Yaskawa INFORM job: s2D_Face_diagonal.JBI

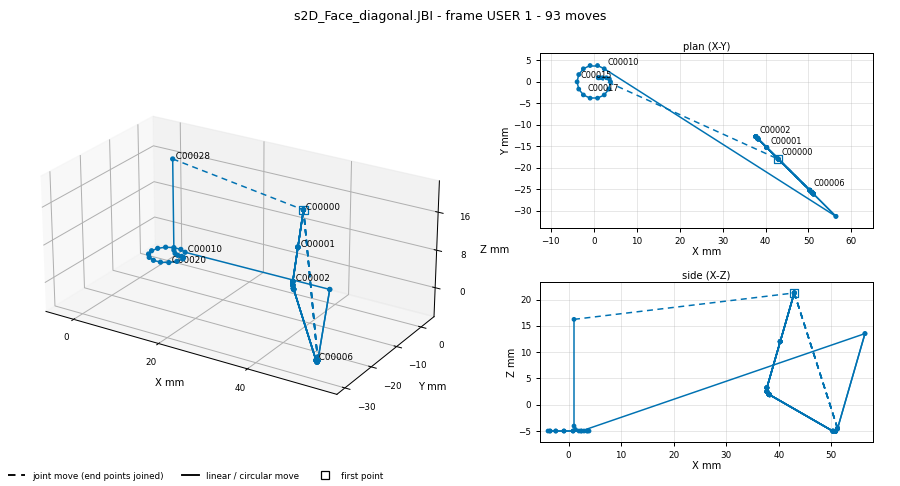
[picture p0: tool path of s2D_Face_diagonal.JBI in frame USER 1, 93 of 93 moves have a stored position in this frame; points joined in program order, loops and branches not executed]
/JOB
//NAME s2D_Face_diagonal
//POS
///NPOS 10,0,0,0,0,0
///USER 1
///TOOL 2
///POSTYPE USER
///RECTAN
///RCONF 1,0,0,0,0,0
C00000=53.984,-29.817,15.539,-90.000,-150.794,-116.565
C00001=53.984,-24.817,6.879,-90.000,-150.794,-116.565
C00002=53.984,-20.744,-0.175,-90.000,-150.794,-116.565
C00003=53.705,-20.407,-0.758,-90.000,-150.794,-116.565
C00004=53.031,-20.268,-1.000,-90.000,-150.794,-116.565
C00005=-55.536,-20.268,-1.000,-90.000,-150.794,-116.565
C00006=-56.209,-20.407,-0.758,-90.000,-150.794,-116.565
C00007=-56.488,-20.744,-0.175,-90.000,-150.794,-116.565
C00008=-56.488,-29.817,15.539,-90.000,-150.794,-116.565
C00000=-54.817,-31.806,15.539,180.000,-152.507,146.310
C00001=-49.817,-31.806,6.879,180.000,-152.507,146.310
C00002=-45.903,-31.806,0.100,180.000,-152.507,146.310
C00003=-45.454,-31.434,-0.678,180.000,-152.507,146.310
C00004=-45.268,-30.536,-1.000,180.000,-152.507,146.310
C00005=-45.268,32.000,-1.000,180.000,-152.507,146.310
C00006=-45.454,32.898,-0.678,180.000,-152.507,146.310
C00007=-45.903,33.270,0.100,180.000,-152.507,146.310
C00008=-54.817,33.270,15.539,180.000,-152.507,146.310
C00000=-54.817,-31.488,15.539,180.000,-152.507,146.310
C00001=-49.817,-31.488,6.879,180.000,-152.507,146.310
C00002=-45.744,-31.488,-0.175,180.000,-152.507,146.310
C00003=-45.407,-31.209,-0.758,180.000,-152.507,146.310
C00004=-45.268,-30.536,-1.000,180.000,-152.507,146.310
C00005=-45.268,32.000,-1.000,180.000,-152.507,146.310
C00006=-45.407,32.674,-0.758,180.000,-152.507,146.310
C00007=-45.744,32.952,-0.175,180.000,-152.507,146.310
C00008=-54.817,32.952,15.539,180.000,-152.507,146.310
C00000=-57.952,29.817,15.539,90.000,-150.794,63.435
C00001=-57.952,24.817,6.879,90.000,-150.794,63.435
C00002=-57.952,20.744,-0.175,90.000,-150.794,63.435
C00003=-57.674,20.407,-0.758,90.000,-150.794,63.435
C00004=-57.000,20.268,-1.000,90.000,-150.794,63.435
C00005=54.657,20.268,-1.000,90.000,-150.794,63.435
C00006=55.330,20.407,-0.758,90.000,-150.794,63.435
C00007=55.609,20.744,-0.175,90.000,-150.794,63.435
C00008=55.609,29.817,15.539,90.000,-150.794,63.435
C00000=-57.952,29.817,15.539,90.000,-150.794,63.435
C00001=-57.952,24.817,6.879,90.000,-150.794,63.435
C00002=-57.952,20.744,-0.175,90.000,-150.794,63.435
C00003=-57.674,20.407,-0.758,90.000,-150.794,63.435
C00004=-57.000,20.268,-1.000,90.000,-150.794,63.435
C00005=54.657,20.268,-1.000,90.000,-150.794,63.435
C00006=55.330,20.407,-0.758,90.000,-150.794,63.435
C00007=55.609,20.744,-0.175,90.000,-150.794,63.435
C00008=55.609,29.817,15.539,90.000,-150.794,63.435
C00000=1.040,-0.952,16.240,0.000,-180.000,-30.000
C00001=1.040,-0.952,6.080,0.000,-180.000,-30.000
C00002=1.040,-0.952,2.000,0.000,-180.000,-30.000
C00003=1.040,-0.952,-4.048,0.000,-180.000,-30.000
C00004=1.319,-0.952,-4.721,0.000,-180.000,-30.000
C00005=1.993,-0.952,-5.000,0.000,-180.000,-30.000
C00006=2.945,-0.952,-5.000,0.000,-180.000,-30.000
C00007=3.619,-0.674,-5.000,0.000,-180.000,-30.000
C00008=3.898,0.000,-5.000,0.000,-180.000,-30.000
C00009=3.512,1.691,-5.000,0.000,-180.000,-30.000
C00010=2.430,3.047,-5.000,0.000,-180.000,-30.000
C00011=0.867,3.800,-5.000,0.000,-180.000,-30.000
C00012=-0.867,3.800,-5.000,0.000,-180.000,-30.000
C00013=-2.430,3.047,-5.000,0.000,-180.000,-30.000
C00014=-3.512,1.691,-5.000,0.000,-180.000,-30.000
C00015=-3.898,0.000,-5.000,0.000,-180.000,-30.000
C00016=-3.512,-1.691,-5.000,0.000,-180.000,-30.000
C00017=-2.430,-3.047,-5.000,0.000,-180.000,-30.000
C00018=-0.867,-3.800,-5.000,0.000,-180.000,-30.000
C00019=0.867,-3.800,-5.000,0.000,-180.000,-30.000
C00020=2.430,-3.047,-5.000,0.000,-180.000,-30.000
C00021=3.512,-1.691,-5.000,0.000,-180.000,-30.000
C00022=3.898,0.000,-5.000,0.000,-180.000,-30.000
C00023=3.619,0.674,-5.000,0.000,-180.000,-30.000
C00024=2.945,0.952,-5.000,0.000,-180.000,-30.000
C00025=1.993,0.952,-5.000,0.000,-180.000,-30.000
C00026=1.319,0.952,-4.721,0.000,-180.000,-30.000
C00027=1.040,0.952,-4.048,0.000,-180.000,-30.000
C00028=1.040,0.952,16.240,0.000,-180.000,-30.000
C00000=54.817,30.609,15.539,0.000,-152.507,-33.690
C00001=49.817,30.609,6.879,0.000,-152.507,-33.690
C00002=45.744,30.609,-0.175,0.000,-152.507,-33.690
C00003=45.407,30.330,-0.758,0.000,-152.507,-33.690
C00004=45.268,29.657,-1.000,0.000,-152.507,-33.690
C00005=45.268,-28.031,-1.000,0.000,-152.507,-33.690
C00006=45.407,-28.705,-0.758,0.000,-152.507,-33.690
C00007=45.744,-28.984,-0.175,0.000,-152.507,-33.690
C00008=54.817,-28.984,15.539,0.000,-152.507,-33.690
C00000=42.939,-17.984,21.265,-45.000,-157.889,-76.068
C00001=40.267,-15.312,12.007,-45.000,-157.889,-76.068
C00002=37.731,-12.775,3.222,-45.000,-157.889,-76.068
C00003=37.734,-12.777,2.493,-45.000,-157.889,-76.068
C00004=38.102,-13.142,1.980,-45.000,-157.889,-76.068
C00005=38.252,-13.291,1.894,-45.000,-157.889,-76.068
C00006=50.300,-25.246,-5.035,-45.000,-157.889,-76.068
C00007=50.818,-25.760,-5.032,-45.000,-157.889,-76.068
C00008=51.181,-26.122,-4.514,-45.000,-157.889,-76.068
C00009=56.390,-31.330,13.530,-45.000,-157.889,-76.068
//INST
///ATTR SC,RW,RJ
////FRAME USER 1
///GROUP1 RB1
///LVARS 2,0,0,0,0,0,0,0
NOP
SET LB000 1
SET LB001 25
MOVJ C00000 VJ=17
MOVL C00001 V=17 PL=LB000 ACC=LB001 DEC=LB001
' Plunge Move Starts
MOVL C00002 V=8 PL=LB000 ACC=LB001 DEC=LB001
' Lead In Move Starts
MOVL C00003 V=17 PL=LB000 ACC=LB001 DEC=LB001
MOVL C00004 V=17 PL=LB000 ACC=LB001 DEC=LB001
' Cutting Move Starts
MOVL C00005 V=17 PL=LB000 ACC=LB001 DEC=LB001
' Lead Out Move Starts
MOVL C00006 V=17 PL=LB000 ACC=LB001 DEC=LB001
MOVL C00007 V=17 PL=LB000 ACC=LB001 DEC=LB001
' Rapid Move Starts
MOVL C00008 V=17 PL=LB000 ACC=LB001 DEC=LB001
' By Autodesk Fusion CAM 2.0.20494
' Tool = 2
' Spindle = 5000 RPM
' Set Position Level
' Set Acceleration
' Program Start
' First Toolpath Point
' Last Toolpath Point
MOVJ C00000 VJ=17
MOVL C00001 V=17 PL=LB000 ACC=LB001 DEC=LB001
' Plunge Move Starts
MOVL C00002 V=8 PL=LB000 ACC=LB001 DEC=LB001
' Lead In Move Starts
MOVL C00003 V=17 PL=LB000 ACC=LB001 DEC=LB001
MOVL C00004 V=17 PL=LB000 ACC=LB001 DEC=LB001
' Cutting Move Starts
MOVL C00005 V=17 PL=LB000 ACC=LB001 DEC=LB001
' Lead Out Move Starts
MOVL C00006 V=17 PL=LB000 ACC=LB001 DEC=LB001
MOVL C00007 V=17 PL=LB000 ACC=LB001 DEC=LB001
' Rapid Move Starts
MOVL C00008 V=17 PL=LB000 ACC=LB001 DEC=LB001
' By Autodesk Fusion CAM 2.0.20494
' Tool = 8
' Spindle = 6000 RPM
' Set Position Level
' Set Acceleration
' Program Start
' First Toolpath Point
' Last Toolpath Point
MOVJ C00000 VJ=17
MOVL C00001 V=17 PL=LB000 ACC=LB001 DEC=LB001
' Plunge Move Starts
MOVL C00002 V=8 PL=LB000 ACC=LB001 DEC=LB001
' Lead In Move Starts
MOVL C00003 V=17 PL=LB000 ACC=LB001 DEC=LB001
MOVL C00004 V=17 PL=LB000 ACC=LB001 DEC=LB001
' Cutting Move Starts
MOVL C00005 V=17 PL=LB000 ACC=LB001 DEC=LB001
' Lead Out Move Starts
MOVL C00006 V=17 PL=LB000 ACC=LB001 DEC=LB001
MOVL C00007 V=17 PL=LB000 ACC=LB001 DEC=LB001
' Rapid Move Starts
MOVL C00008 V=17 PL=LB000 ACC=LB001 DEC=LB001
' By Autodesk Fusion CAM 2.0.20494
' Tool = 2
' Spindle = 5000 RPM
' Set Position Level
' Set Acceleration
' Program Start
' First Toolpath Point
' Last Toolpath Point
MOVJ C00000 VJ=17
MOVL C00001 V=17 PL=LB000 ACC=LB001 DEC=LB001
' Plunge Move Starts
MOVL C00002 V=8 PL=LB000 ACC=LB001 DEC=LB001
' Lead In Move Starts
MOVL C00003 V=17 PL=LB000 ACC=LB001 DEC=LB001
MOVL C00004 V=17 PL=LB000 ACC=LB001 DEC=LB001
' Cutting Move Starts
MOVL C00005 V=17 PL=LB000 ACC=LB001 DEC=LB001
' Lead Out Move Starts
MOVL C00006 V=17 PL=LB000 ACC=LB001 DEC=LB001
MOVL C00007 V=17 PL=LB000 ACC=LB001 DEC=LB001
' Rapid Move Starts
MOVL C00008 V=17 PL=LB000 ACC=LB001 DEC=LB001
' By Autodesk Fusion CAM 2.0.20494
' Tool = 2
' Spindle = 5000 RPM
' Set Position Level
' Set Acceleration
' Program Start
' First Toolpath Point
' Last Toolpath Point
MOVJ C00000 VJ=17
MOVL C00001 V=17 PL=LB000 ACC=LB001 DEC=LB001
' Plunge Move Starts
MOVL C00002 V=8 PL=LB000 ACC=LB001 DEC=LB001
' Lead In Move Starts
MOVL C00003 V=17 PL=LB000 ACC=LB001 DEC=LB001
MOVL C00004 V=17 PL=LB000 ACC=LB001 DEC=LB001
' Cutting Move Starts
MOVL C00005 V=17 PL=LB000 ACC=LB001 DEC=LB001
' Lead Out Move Starts
MOVL C00006 V=17 PL=LB000 ACC=LB001 DEC=LB001
MOVL C00007 V=17 PL=LB000 ACC=LB001 DEC=LB001
' Rapid Move Starts
MOVL C00008 V=17 PL=LB000 ACC=LB001 DEC=LB001
' By Autodesk Fusion CAM 2.0.20494
' Tool = 2
' Spindle = 5000 RPM
' Set Position Level
' Set Acceleration
' Program Start
' First Toolpath Point
' Last Toolpath Point
MOVJ C00000 VJ=17
MOVL C00001 V=17 PL=LB000 ACC=LB001 DEC=LB001
' Plunge Move Starts
MOVL C00002 V=8 PL=LB000 ACC=LB001 DEC=LB001
MOVL C00003 V=8 PL=LB000 ACC=LB001 DEC=LB001
' Lead In Move Starts
MOVL C00004 V=17 PL=LB000 ACC=LB001 DEC=LB001
MOVL C00005 V=17 PL=LB000 ACC=LB001 DEC=LB001
MOVL C00006 V=17 PL=LB000 ACC=LB001 DEC=LB001
MOVL C00007 V=17 PL=LB000 ACC=LB001 DEC=LB001
MOVL C00008 V=17 PL=LB000 ACC=LB001 DEC=LB001
' Cutting Move Starts
MOVL C00009 V=17 PL=LB000 ACC=LB001 DEC=LB001
MOVL C00010 V=17 PL=LB000 ACC=LB001 DEC=LB001
MOVL C00011 V=17 PL=LB000 ACC=LB001 DEC=LB001
MOVL C00012 V=17 PL=LB000 ACC=LB001 DEC=LB001
MOVL C00013 V=17 PL=LB000 ACC=LB001 DEC=LB001
MOVL C00014 V=17 PL=LB000 ACC=LB001 DEC=LB001
MOVL C00015 V=17 PL=LB000 ACC=LB001 DEC=LB001
MOVL C00016 V=17 PL=LB000 ACC=LB001 DEC=LB001
MOVL C00017 V=17 PL=LB000 ACC=LB001 DEC=LB001
MOVL C00018 V=17 PL=LB000 ACC=LB001 DEC=LB001
MOVL C00019 V=17 PL=LB000 ACC=LB001 DEC=LB001
MOVL C00020 V=17 PL=LB000 ACC=LB001 DEC=LB001
MOVL C00021 V=17 PL=LB000 ACC=LB001 DEC=LB001
MOVL C00022 V=17 PL=LB000 ACC=LB001 DEC=LB001
' Lead Out Move Starts
MOVL C00023 V=17 PL=LB000 ACC=LB001 DEC=LB001
MOVL C00024 V=17 PL=LB000 ACC=LB001 DEC=LB001
MOVL C00025 V=17 PL=LB000 ACC=LB001 DEC=LB001
MOVL C00026 V=17 PL=LB000 ACC=LB001 DEC=LB001
MOVL C00027 V=17 PL=LB000 ACC=LB001 DEC=LB001
' Rapid Move Starts
MOVL C00028 V=17 PL=LB000 ACC=LB001 DEC=LB001
' By Autodesk Fusion CAM 2.0.20494
' Tool = 2
' Spindle = 5000 RPM
' Set Position Level
' Set Acceleration
' Program Start
' First Toolpath Point
' Last Toolpath Point
MOVJ C00000 VJ=17
MOVL C00001 V=17 PL=LB000 ACC=LB001 DEC=LB001
' Plunge Move Starts
MOVL C00002 V=8 PL=LB000 ACC=LB001 DEC=LB001
' Lead In Move Starts
MOVL C00003 V=17 PL=LB000 ACC=LB001 DEC=LB001
MOVL C00004 V=17 PL=LB000 ACC=LB001 DEC=LB001
' Cutting Move Starts
MOVL C00005 V=17 PL=LB000 ACC=LB001 DEC=LB001
' Lead Out Move Starts
MOVL C00006 V=17 PL=LB000 ACC=LB001 DEC=LB001
MOVL C00007 V=17 PL=LB000 ACC=LB001 DEC=LB001
' Rapid Move Starts
MOVL C00008 V=17 PL=LB000 ACC=LB001 DEC=LB001
' By Autodesk Fusion CAM 2.0.20494
' Tool = 2
' Spindle = 5000 RPM
' Set Position Level
' Set Acceleration
' Program Start
' First Toolpath Point
' Last Toolpath Point
MOVJ C00000 VJ=17
MOVL C00001 V=17 PL=LB000 ACC=LB001 DEC=LB001
' Plunge Move Starts
MOVL C00002 V=8 PL=LB000 ACC=LB001 DEC=LB001
' Lead In Move Starts
MOVL C00003 V=17 PL=LB000 ACC=LB001 DEC=LB001
MOVL C00004 V=17 PL=LB000 ACC=LB001 DEC=LB001
MOVL C00005 V=17 PL=LB000 ACC=LB001 DEC=LB001
' Cutting Move Starts
MOVL C00006 V=17 PL=LB000 ACC=LB001 DEC=LB001
' Lead Out Move Starts
MOVL C00007 V=17 PL=LB000 ACC=LB001 DEC=LB001
MOVL C00008 V=17 PL=LB000 ACC=LB001 DEC=LB001
' Rapid Move Starts
MOVL C00009 V=17 PL=LB000 ACC=LB001 DEC=LB001
' By Autodesk Fusion CAM 2.0.20494
' Tool = 2
' Spindle = 5000 RPM
' Set Position Level
' Set Acceleration
' Program Start
' First Toolpath Point
END
